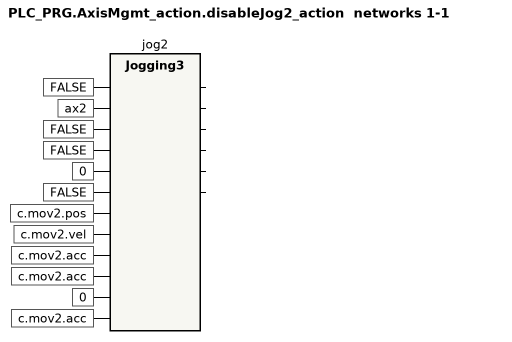
[picture p24: PLC_PRG.AxisMgmt_action.disableJog2_action (FBD) networks 1-1]
_FBD_ (* Function Block Diagram *)
NETWORK 1
	jog2:Jogging3(FALSE, ax2, FALSE, FALSE, 0, FALSE, c.mov2.pos, c.mov2.vel, c.mov2.acc, c.mov2.acc, 0, c.mov2.acc)
_END_FBD_
(* the same logic as Structured Text *)
(* Network 1 *)
jog2(FALSE, ax2, FALSE, FALSE, 0, FALSE, c.mov2.pos, c.mov2.vel, c.mov2.acc, c.mov2.acc, 0, c.mov2.acc);
END_ACTION

ACTION updateRelTapePos_entry:
flagProcessingPack:=TRUE;
END_ACTION

ACTION updateRelTapePos_action:
IF ( tape.Position > tape_pos_off ) THEN
	tape_pos_rel :=tape.Position -tape_pos_off;
ELSE
	tape_pos_rel :=tape.Position -tape_pos_off + c.tape.period;
END_IF

IF ( tape_pos_rel>c.tape.period-10 ) THEN
	flagProcessingPack:=FALSE;
END_IF
END_ACTION

ACTION signalTimeOut_action:
tapeTimedOut:=TRUE;
END_ACTION

ACTION stopTape_action:
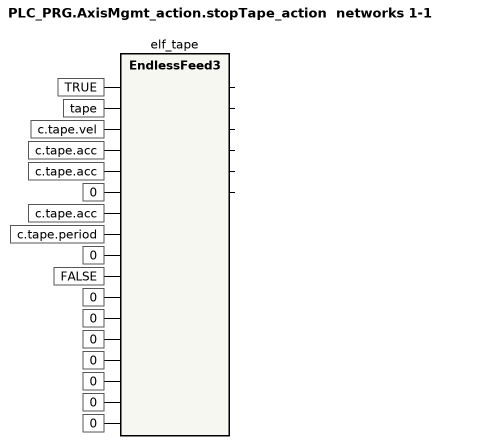
_FBD_ (* Function Block Diagram *)
NETWORK 1
	elf_tape:EndlessFeed3(TRUE, tape, c.tape.vel, c.tape.acc, c.tape.acc, 0, c.tape.acc, c.tape.period, 0, FALSE, 0, 0, 0, 0, 0, 0, 0)
_END_FBD_
(* the same logic as Structured Text *)
(* Network 1 *)
elf_tape(TRUE, tape, c.tape.vel, c.tape.acc, c.tape.acc, 0, c.tape.acc, c.tape.period, 0, FALSE, 0, 0, 0, 0, 0, 0, 0);
END_ACTION

ACTION disableTape_action:
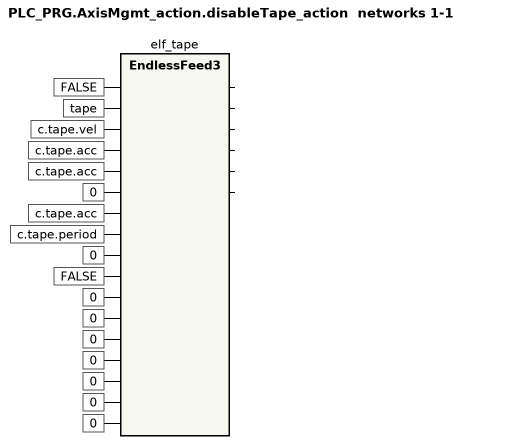
_FBD_ (* Function Block Diagram *)
NETWORK 1
	elf_tape:EndlessFeed3(FALSE, tape, c.tape.vel, c.tape.acc, c.tape.acc, 0, c.tape.acc, c.tape.period, 0, FALSE, 0, 0, 0, 0, 0, 0, 0)
_END_FBD_
(* the same logic as Structured Text *)
(* Network 1 *)
elf_tape(FALSE, tape, c.tape.vel, c.tape.acc, c.tape.acc, 0, c.tape.acc, c.tape.period, 0, FALSE, 0, 0, 0, 0, 0, 0, 0);
END_ACTION

ACTION signalSyncStop_action:
syncStopOk:=TRUE;
END_ACTION
END_ACTION

ACTION OpModeMgmt_action:
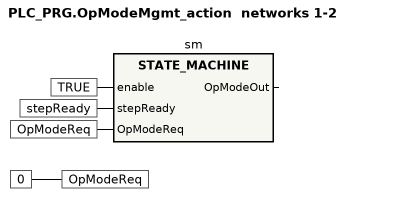
_FBD_ (* Function Block Diagram *)
NETWORK 1
	sm:STATE_MACHINE(enable: TRUE, stepReady: stepReady, OpModeReq: OpModeReq)
NETWORK 2
	0 => OpModeReq
_END_FBD_
(* the same logic as Structured Text *)
(* Network 1 *)
sm(enable := TRUE, stepReady := stepReady, OpModeReq := OpModeReq);
(* Network 2 *)
OpModeReq := 0;
END_ACTION
END_PROGRAM

(* POU STATE_MACHINE, ST *)
FUNCTION_BLOCK STATE_MACHINE
VAR
	InternalState:INT:=0;
	flagEnable:BOOL:=0;
END_VAR
VAR_INPUT
	enable:BOOL;
	stepReady:BOOL;
	OpModeReq:INT;
END_VAR
VAR_OUTPUT
	OpModeOut:INT:=0;
END_VAR
IF ( NOT enable ) THEN
	InternalState:=0;
	flagEnable:=FALSE;
	OpModeOut:=0;
	RETURN;
END_IF
flagEnable:=TRUE;

CASE InternalState OF
10: (* disabling... *)
	IF (  stepReady ) THEN	(* disable ok *)
		InternalState:=15;
		OpModeOut:=0;
	END_IF
15: (*disabled, waiting for enable *)
	IF ( OpModeReq=20 ) THEN
		OpModeOut:=20;
		InternalState:=20;
	ELSE
		OpModeOut:=0;
	END_IF
20: (* enabling *)
	IF ( StepReady ) THEN (* enabling completed *)
		InternalState:=25;
		OpModeOut:=0;
	END_IF
25: (*enabled: waiting for disable or homing*)
	IF ( OpModeReq = 10 ) THEN
		OpModeOut:=10;
		InternalState:=10;
	ELSIF ( OpModeReq = 30 ) THEN
		OpModeOut:=30;
		InternalState:=30;
	ELSIF ( OpModeReq = 40 ) THEN (* FIXME this should not be enabled *)
		OpModeOut:=40;
		InternalState:=40;
	END_IF
30:
	IF (  stepReady ) THEN (* homing completed *)
		InternalState:=35;
		OpModeOut:=0;
	END_IF
35: (* Homed, waiting for disable or auto *)
	IF ( OpModeReq = 10 ) THEN
		InternalState:=10;
		OpModeOut:=10;
	ELSIF ( OpModeReq = 40 ) THEN
		InternalState:=40;
	END_IF
40: (* in auto mode *)
	OpModeOut:=40;
	IF ( OpModeReq=50 ) THEN (* auto mode started *)
		InternalState:=50;
	END_IF
50:	(* syncStop-ing *)
	OpModeOut:=50;
	IF ( stepReady ) THEN (* stopping completed *)
		InternalState:=55;
	END_IF
55: (* stopped,waiting for auto or disable*)
	OpModeOut:=0;
	IF ( OpModeReq = 10 ) THEN
		InternalState:=10;
		OpModeOut:=10;
	ELSIF ( OpModeReq = 40 ) THEN
		InternalState:=40;
		OpModeOut:=40;
	END_IF
ELSE
	InternalState:=10;
	OpModeOut:=10;
END_CASE
END_FUNCTION_BLOCK
